{attribute 'linkalways'} 
{attribute 'no_explicit_call' := 'This FB is a CLASS and must be accessed using methods or properties'}
{attribute 'enable_dynamic_creation'}
FUNCTION_BLOCK FINAL SEL_UINT EXTENDS Node
VAR
	g : _BOOL(FALSE);
	in1 : _UINT(0);
	in2 : _UINT(0);
	out : _UINT(0);
END_VAR

METHOD PUBLIC Clone : I_Node
VAR
	pNode : POINTER TO SEL_UINT;
END_VAR
pNode := __NEW(SEL_UINT);
Clone := pNode^;
END_METHOD

METHOD FB_init : BOOL
VAR_INPUT
	bInitRetains : BOOL; // if TRUE, the retain variables are initialized (warm start / cold start)
	bInCopyCode : BOOL;  // if TRUE, the instance afterwards gets moved into the copy code (online change)
END_VAR
AddInput('g',THIS^.g);
AddInput('in1',THIS^.in1);
AddInput('in2',THIS^.in2);
AddOutput('out', THIS^.out);
END_METHOD

METHOD PROTECTED OnExecute
VAR
END_VAR
IF g.value THEN
	out.value := in2.value;
ELSE
	out.value := in1.value;
END_IF
END_METHOD

END_FUNCTION_BLOCK

(* stored: Version 1.1.0.1, ProductVersion 3.1.4024.15
   POU SEL_UINT: Id {a9921843-e418-4d60-9c4d-53d1c68aa2c1}, SpecialFunc None
   Folder Constructor: Id {0fe7985e-c839-4247-83be-8b6f6dd6b0f1}
   Method Clone: Id {480c57b4-0812-4047-86ba-fe62232d0336}
   Method FB_init: Id {aac259e8-ee7f-405f-9e19-3c3805e317bc}
   Method OnExecute: Id {f18ab8b6-1468-40df-be88-07d51d9b3fad} *)
